{attribute addProperty BoxType "IODEVICETYPE_ETHERCATPROT"}
{attribute addProperty Id "boxesboxes_B14E9406325274065.875A_0076_AMP8000_0030_0103AMP8000_5E0E86F855669.5SyncUnitsSyncUnits_CAB22D3B19524.375InputsInputs_C75D3FEC1280160OutputsOutputs_47D1E803848106InfoDataInfoData_E9F65A829612"}
{attribute addProperty CRC "4281505233"}
{attribute addProperty SizeInBites "35502"}
{attribute addProperty SizeInBytes "4437.75"}
TYPE EtherCAT_Master_Duplicates_FF3295D1 :
STRUCT
	{attribute addProperty Name "boxes"}
	boxes : boxes_B14E9406;
	{attribute addProperty Name "A_0076_AMP8000_0030_0103"}
	A_0076_AMP8000_0030_0103 : AMP8000_5E0E86F8;
	{attribute addProperty Name "SyncUnits"}
	SyncUnits : SyncUnits_CAB22D3B;
	{attribute addProperty Name "Inputs"}
	Inputs : Inputs_C75D3FEC;
	{attribute addProperty Name "Outputs"}
	Outputs : Outputs_47D1E803;
	{attribute addProperty Name "InfoData"}
	InfoData : InfoData_E9F65A82;
END_STRUCT
END_TYPE

(* stored: Version 1.2.0.0, ProductVersion 3.1.4024.9
   DUT EtherCAT_Master_Duplicates_FF3295D1: Id {ff3c6d05-3938-40c9-8874-0470cee1e04f} *)
